TYPE ST_1:
STRUCT
	sStruct : ST_2;
	sstring : STRING(80);
END_STRUCT
END_TYPE

(* stored: Version 1.1.0.1, ProductVersion 3.1.4024.12
   DUT ST_1: Id {9e592088-2333-48a3-955b-1540c5c00897} *)
